{attribute 'qualified_only'}
{attribute 'strict'}
TYPE eTcoMitsubishiRoboticsSimpleTests : (
    Restore := 1,
    CleanUp,
    Message,
    PowerDisable,
    PowerEnable,
    Reset,
    MoveRelativePositiveWithDisabledPositiveDirection,
    MoveRelativePositiveWithEnabledPositiveDirection,
    MoveRelativeNegativeWithDisabledNegativeDirection,
    MoveRelativeNegativeWithEnabledNegativeDirection,
    HommingDirect,
    MoveVelocityPositiveWithDisabledPositiveDirection,
    MoveVelocityPositiveWithEnabledPositiveDirection,
    Stop,
    MoveVelocityNegativeWithDisabledNegativeDirection,
    MoveVelocityNegativeWithEnabledNegativeDirection,
    MoveAbsoluteDisabled,
    MoveAbsoluteDisabledPositiveDirection,
    MoveAbsoluteEnabledPositiveDirection,
    MoveAbsoluteDisabledNegativeDirection,
    MoveAbsoluteEnabledNegativeDirection,
    Last
);
END_TYPE

(* stored: Version 1.1.0.1, ProductVersion 3.1.4024.12
   DUT eTcoMitsubishiRoboticsSimpleTests: Id {175cfec2-27d0-0a24-0958-a7809ba4f177} *)
